FUNCTION_BLOCK Aborted_State IMPLEMENTS ITF_State
VAR_INPUT
END_VAR
VAR_OUTPUT
END_VAR
VAR
	pPML_Base : POINTER TO PML_Base;
	_stateMachine : IPmlStateMachine;
	bClear : BOOL;
END_VAR

METHOD Cycle : BOOL
VAR_INPUT
END_VAR
IF bClear THEN
	pPML_Base^.SetState(pPML_Base^.clearing);
	_stateMachine.PMLCommand(Command := E_PMLCommand.ePMLCommand_Clear);
END_IF
END_METHOD

METHOD FB_init : BOOL
VAR_INPUT
	bInitRetains : BOOL; // if TRUE, the retain variables are initialized (warm start / cold start)
	bInCopyCode : BOOL;  // if TRUE, the instance afterwards gets moved into the copy code (online change)
	pPML_Base : POINTER TO PML_Base;
	statemachine : IPmlStateMachine;
END_VAR
_stateMachine := statemachine;
THIS^.pPML_Base := pPML_Base;
END_METHOD

END_FUNCTION_BLOCK

(* stored: Version 1.1.0.1, ProductVersion 3.1.4024.11
   POU Aborted_State: Id {7558cd23-d105-48b5-ae40-6c8d917c4b3e}, SpecialFunc None
   Method Cycle: Id {fd45476c-1766-427a-ba07-14844846e329}
   Method FB_init: Id {76d2174b-6217-4d54-8806-813df1582835} *)
